FUNCTION_BLOCK FB_HomeVirtual
VAR_INPUT
	En: BOOL;
	bReset: BOOL;
	bExecute: BOOL;
	nCmdData: UINT;
	bLimitFwd: BOOL;
	bLimitBwd: BOOL;	
	bHomeSensor: BOOL;	
	fHomePosition:LREAL;
	nHomeRevOffset: UINT;
END_VAR
VAR_IN_OUT
	Axis: AXIS_REF;
END_VAR
VAR_OUTPUT
	EnO: BOOL;	
	bBusy: BOOL;
	bDone: BOOL;
	bHomed:BOOL;
	bError: BOOL;
	nErrorId: UDINT;
END_VAR
VAR
	fbHomeToSwitch: FB_HomeToSwitch;
    fbHomeDirect: FB_HomeDirect; //Only used for direct homing (set of position)
    fbMoveVelocity:MC_MoveVelocity;
	fbHomeReadNCVelocities: FB_HomeReadNcVelocities;	
    fbHomeReset:MC_Home;   //Only used for reset of calibration flag		
	fbExecuteRiseEdge: R_TRIG;
	fbExecuteFallEdge: F_TRIG;
	nHomingState:INT:=0;
	bExecuteHomeToSwitch:BOOL:=FALSE;
	bExecuteMoveVelocity:BOOL:=FALSE;
	bExecuteReadNCVelocities: BOOL:=FALSE;
	bSequenceReady:BOOL:=TRUE;
	fVelocityToCamNC: LREAL;
	fVelocityFromCamNC: LREAL;	
	bExecuteMCHome:BOOL:=FALSE;
	bNCVelocitiesReadOnce:BOOL:=FALSE;	
	bExecuteHomeDirect: BOOL;
	bNCVelocitiesCorrupted:BOOL:=FALSE;
	nCmdDataLocal: UINT;  //Ensure that nCmdData is not changed during sequence
END_VAR

EnO:=En;

IF bReset THEN	
	bError:=FALSE;
	nErrorId:=0;
END_IF

// Reset when bExecute is low
IF NOT bExecute THEN
  nHomingState:=0;
  bSequenceReady:=TRUE;
  bExecuteHomeToSwitch:=FALSE;
  bExecuteHomeDirect:=FALSE;
  bExecuteMCHome:=FALSE;
  bExecuteMoveVelocity:=FALSE;
  bExecuteReadNCVelocities:=FALSE;
END_IF

//Reset at rinsing edge of bExecute
fbExecuteRiseEdge(CLK:=bExecute);
IF fbExecuteRiseEdge.Q THEN
  nCmdDataLocal:=nCmdData; //Ensure that nCmdData is not changed during sequence (nCmdData will only be read at a rising edge of bExecute)
  bNCVelocitiesCorrupted:=FALSE;
  bSequenceReady:=FALSE;
  bExecuteReadNCVelocities:=NOT(nCmdDataLocal=15);  // Not needed for sequence 15 (set position only, no movement))  
  bExecuteMCHome:=TRUE;
  //Check if valid nCmdDataLocal
  CASE nCmdDataLocal OF  	
    1:
    2:
    3:
    4:
    15:
    ELSE //nCmdData not valid	
      bError:=TRUE;
      nErrorId:=16#4FFF;   
  END_CASE
END_IF

// Read NC homing velocities at bExecute rising edge
fbHomeReadNCVelocities(
  En:=En,
  bExecute:=bExecuteReadNCVelocities,
  bReset:=bReset,
  Axis:=Axis,
);

IF fbHomeReadNCVelocities.bDone THEN
  	fVelocityFromCamNC:=fbHomeReadNCVelocities.fVelocityFromCam;
    fVelocityToCamNC:=fbHomeReadNCVelocities.fVelocityToCam;
	bNCVelocitiesReadOnce:=TRUE;  //Allow write back of homing velocities
	bExecuteReadNCVelocities:=FALSE;
END_IF

//Homing Sequences
CASE nCmdDataLocal OF  
	
   1: // Home to low limit switch
	   CASE nHomingState OF
		  0:
		    bHomed:=Axis.Status.Homed;
            // Wait for read of velocities from NC
	        IF fbHomeReadNCVelocities.bDone AND fbHomeReset.Done AND bExecute AND NOT bSequenceReady THEN
			  IF bLimitBwd THEN
                nHomingState:=1;
              ELSE
				nHomingState:=2;  //Standing on limit switch go direct to state 2 
              END_IF                                          		  
	        END_IF
		  1: // wait for reach low limit then trigger fbHomeToSwitch
		    bHomed:=FALSE;
			bSequenceReady:=FALSE;
			fbMoveVelocity.Velocity:=ABS(fVelocityToCamNC);
            fbMoveVelocity.Direction:=MC_Negative_Direction;
	        bExecuteMoveVelocity:=bExecute;  // Execute MC_MoveVelocity
		    IF NOT bLimitBwd AND NOT fbMoveVelocity.Busy AND Axis.Status.NotMoving THEN //MC_MoveVelocity.Busy goes down when ramp down initiates (not ends).
			  nHomingState:=2;
		    END_IF
		  2: // Wait for fbHomeToSwitch
		    bHomed:=FALSE;
		    bSequenceReady:=FALSE;
            bExecuteMoveVelocity:=FALSE;			
            bExecuteHomeToSwitch:=TRUE;	
            fbHomeToSwitch.nSearchDirTwoardsCam:=MC_Positive_Direction;
            fbHomeToSwitch.nSearchDirOffCam:=MC_Positive_Direction;	             
	        fbHomeToSwitch.fVelocityToCamNC:=fVelocityToCamNC; // High speed
  	        fbHomeToSwitch.fVelocityFromCamNC:=fVelocityFromCamNC;  // Low speed              		
		    fbHomeToSwitch.bCamSensor:=NOT bLimitBwd;            	 		    
	        IF fbHomeToSwitch.bDone THEN
	          bSequenceReady:=TRUE;
			  nHomingState:=0;
			  bHomed:=Axis.Status.Homed;
	        END_IF;	  		  
	   END_CASE;
		  	  
   2:  // Home to high limit switch
       CASE nHomingState OF      	   
		  0:
		    bHomed:=Axis.Status.Homed;
            // Wait for read of velocities from NC
	        IF fbHomeReadNCVelocities.bDone AND fbHomeReset.Done AND bExecute AND NOT bSequenceReady THEN
			  IF bLimitFwd THEN
                nHomingState:=1;
              ELSE
				nHomingState:=2;  //Standing on limit switch go direct to state 2 
              END_IF                                          		  
	        END_IF
		  1: // wait for reach low limit then trigger fbHomeToSwitch
		    bHomed:=FALSE;
			bSequenceReady:=FALSE;
			fbMoveVelocity.Velocity:=ABS(fVelocityToCamNC);
            fbMoveVelocity.Direction:=MC_Positive_Direction;
	        bExecuteMoveVelocity:=bExecute;  // Execute MC_MoveVelocity
		    IF NOT bLimitFwd AND NOT fbMoveVelocity.Busy AND Axis.Status.NotMoving THEN //MC_MoveVelocity.Busy goes down when ramp down initiates (not ends).
			  nHomingState:=2;
		    END_IF
		  2: // Wait for fbHomeToSwitch
		    bHomed:=FALSE;
		    bSequenceReady:=FALSE;
            bExecuteMoveVelocity:=FALSE;			
            bExecuteHomeToSwitch:=TRUE;	
            fbHomeToSwitch.nSearchDirTwoardsCam:=MC_Negative_Direction;
            fbHomeToSwitch.nSearchDirOffCam:=MC_Negative_Direction;	             
	        fbHomeToSwitch.fVelocityToCamNC:=fVelocityToCamNC; // High speed
  	        fbHomeToSwitch.fVelocityFromCamNC:=fVelocityFromCamNC;  // Low speed              		
		    fbHomeToSwitch.bCamSensor:=NOT bLimitFwd;            	 		    
	        IF fbHomeToSwitch.bDone THEN
	          bSequenceReady:=TRUE;
			  nHomingState:=0;
			  bHomed:=Axis.Status.Homed;
	        END_IF;	  			  
	   END_CASE;
	  
   3:  // Home on bHomeSensor via bLimitBwd
      CASE nHomingState OF
		  0:
		    bHomed:=Axis.Status.Homed;
            // Wait for read of velocities from NC
	        IF fbHomeReadNCVelocities.bDone AND fbHomeReset.Done AND bExecute AND NOT bSequenceReady THEN
			  IF bLimitBwd THEN
                nHomingState:=1;
              ELSE
				nHomingState:=2;  //Standing on limit switch go direct to state 2 
              END_IF                                          		  
	        END_IF
		  1: // wait for reach low limit then trigger fbHomeToSwitch
		    bHomed:=FALSE;
			bSequenceReady:=FALSE;
			fbMoveVelocity.Velocity:=ABS(fVelocityToCamNC);
            fbMoveVelocity.Direction:=MC_Negative_Direction;
	        bExecuteMoveVelocity:=bExecute;  // Execute MC_MoveVelocity
		    IF NOT bLimitBwd AND NOT fbMoveVelocity.Busy AND Axis.Status.NotMoving THEN //MC_MoveVelocity.Busy goes down when ramp down initiates (not ends).
			  nHomingState:=2;
		    END_IF
		  2: // Home to bHomeSensor switch
		    bHomed:=FALSE;
			bSequenceReady:=FALSE;
			bExecuteMoveVelocity:=FALSE;			
            bExecuteHomeToSwitch:=TRUE; 
			fbHomeToSwitch.bCamSensor:=bHomeSensor;
			fbHomeToSwitch.nSearchDirTwoardsCam:=MC_Positive_Direction;
      		fbHomeToSwitch.nSearchDirOffCam:=MC_Positive_Direction;	 
            fbHomeToSwitch.fVelocityToCamNC:=fVelocityToCamNC; // High speed
  	        fbHomeToSwitch.fVelocityFromCamNC:=fVelocityFromCamNC;  // Low speed (restored) 
            IF fbHomeToSwitch.bDone THEN
  			  bNCVelocitiesCorrupted:=FALSE;  //Correct velocities in NC
			  nHomingState:=0;
			  bExecuteHomeToSwitch:=FALSE;
			  bHomed:=Axis.Status.Homed;
			  bSequenceReady:=TRUE;	
            END_IF
	  END_CASE	  
   4: // Home on bHomeSensor via bLimitFwd
       CASE nHomingState OF		   
		  0:
		    bHomed:=Axis.Status.Homed;
            // Wait for read of velocities from NC
	        IF fbHomeReadNCVelocities.bDone AND fbHomeReset.Done AND bExecute AND NOT bSequenceReady THEN
			  IF bLimitFwd THEN
                nHomingState:=1;
              ELSE
				nHomingState:=2;  //Standing on limit switch go direct to state 2 
              END_IF                                          		  
	        END_IF
		  1: // wait for reach low limit then trigger fbHomeToSwitch
		    bHomed:=FALSE;
			bSequenceReady:=FALSE;
			fbMoveVelocity.Velocity:=ABS(fVelocityToCamNC);
            fbMoveVelocity.Direction:=MC_Positive_Direction;
	        bExecuteMoveVelocity:=bExecute;  // Execute MC_MoveVelocity
		    IF NOT bLimitFwd AND NOT fbMoveVelocity.Busy AND Axis.Status.NotMoving THEN //MC_MoveVelocity.Busy goes down when ramp down initiates (not ends).
			  nHomingState:=2;
		    END_IF
		  2: // Home to bHomeSensor switch
		    bHomed:=FALSE;
			bSequenceReady:=FALSE;
			bExecuteMoveVelocity:=FALSE;			
            bExecuteHomeToSwitch:=TRUE; 			
			fbHomeToSwitch.nSearchDirTwoardsCam:=MC_Negative_Direction;
      		fbHomeToSwitch.nSearchDirOffCam:=MC_Negative_Direction;	 
      		fbHomeToSwitch.bCamSensor:=bHomeSensor;
            fbHomeToSwitch.fVelocityToCamNC:=fVelocityToCamNC; // High speed
  	        fbHomeToSwitch.fVelocityFromCamNC:=fVelocityFromCamNC;  // Low speed (restored) 
            IF fbHomeToSwitch.bDone THEN
  			  bNCVelocitiesCorrupted:=FALSE;  //Correct velocities in NC
			  nHomingState:=0;
			  bExecuteHomeToSwitch:=FALSE;
			  bHomed:=Axis.Status.Homed;
			  bSequenceReady:=TRUE;	
            END_IF		  		  
	  END_CASE	  
	  
   15: //Set current position (simplest homing sequence)
     bExecuteHomeDirect:=bExecute;
	 bHomed:=Axis.Status.Homed;
     IF fbHomeDirect.bDone THEN  //Homing ready				
	   bExecuteHomeDirect:=FALSE;				
       bSequenceReady:=TRUE;	
     END_IF
	 bNCVelocitiesCorrupted:=FALSE; // no changes of NC velocities (no restore needed)
	 
ELSE
  fbHomeToSwitch.bCamSensor:=FALSE;
  bHomed:=Axis.Status.Homed;
END_CASE;

//Reset calibration flag
fbHomeReset(
 Execute:=bExecuteMCHome AND bExecute AND NOT bError,
 HomingMode:=MC_ResetCalibration,
 Axis:=Axis
);

// Main homing block
fbHomeToSwitch(
	bExecute:=bExecuteHomeToSwitch AND bExecute AND NOT bError AND NOT bExecuteHomeDirect AND NOT bExecuteMoveVelocity,
 	bReset:=bReset,
	fHomePosition:=fHomePosition,
	Axis:=Axis
);

fbMoveVelocity(
    Execute:= bExecuteMoveVelocity AND bExecute AND NOT bError AND NOT bExecuteHomeToSwitch AND NOT bExecuteHomeDirect,
    Axis:=Axis
);

// No sequence, just set position value (nCmdDataLocal=15). Can not run if fbHomeToSwitch is executed
fbHomeDirect(
	bExecute:=bExecuteHomeDirect AND bExecute AND NOT bError  AND NOT bExecuteHomeToSwitch AND NOT bExecuteMoveVelocity,
 	bReset:=bReset,
	fHomePosition:=fHomePosition,
	Axis:=Axis
);

// Error handling
IF NOT bError THEN
  IF fbHomeToSwitch.bError THEN 
	bError:=fbHomeToSwitch.bError;
	nErrorId:=fbHomeToSwitch.nErrorId;
  ELSIF fbHomeReadNCVelocities.bError THEN
	bError:=fbHomeReadNCVelocities.bError;
	nErrorId:=fbHomeReadNCVelocities.nErrorId;
  ELSIF fbHomeDirect.bError THEN
	bError:=fbHomeDirect.bError;
	nErrorId:=fbHomeDirect.nErrorId;
  ELSIF fbMoveVelocity.Error THEN
	bError:=fbMoveVelocity.Error;
	nErrorId:=fbMoveVelocity.ErrorId;    		    		
  END_IF;	
END_IF

// Done and busy bit
bDone:=bSequenceReady AND bExecute;
bBusy:=NOT bSequenceReady;	 

RETURN;

END_FUNCTION_BLOCK

(* stored: Version 1.1.0.1, ProductVersion 3.1.4022.6
   POU FB_HomeVirtual: Id {a69b16ef-d088-4494-bcb3-4c391e3a9c2d}, SpecialFunc None *)
